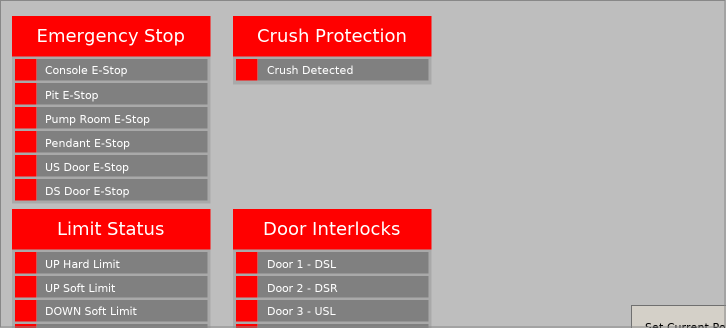
VISUALIZATION SAFETY_PANEL  // 726x328
    Rectangle (233,39 198x45)
    Rectangle (12,38 198x165)
    Rectangle (233,228 198x120)
    Rectangle (12,228 198x144)
    RoundedRectangle (15,276 21x21), colour toggle: HMI.bSoftUpLimFlag
    Rectangle (37,276 170x21)
    Rectangle (42,275 130x27), "UP Soft Limit"
    RoundedRectangle (15,300 21x21), colour toggle: HMI.bSoftDownLimFlag
    Rectangle (37,300 170x21)
    Rectangle (42,298 130x27), "DOWN Soft Limit"
    RoundedRectangle (15,324 21x21), colour variable: HMI_Hard_Limits.DownHardLimit
    Rectangle (37,324 170x21)
    Rectangle (42,322 130x27), "DOWN Hard Limit"
    RoundedRectangle (12,209 198x40), "Limit Status", colour toggle: HMI.bLimitHeaderFlag
    RoundedRectangle (236,252 21x21), colour variable: HMI_Door_Toggle.dwDoor1
    Rectangle (258,252 170x21)
    Rectangle (264,251 130x27), "Door 1 - DSL"
    RoundedRectangle (236,276 21x21), colour variable: HMI_Door_Toggle.dwDoor2
    Rectangle (258,276 170x21)
    Rectangle (264,275 130x27), "Door 2 - DSR"
    RoundedRectangle (236,300 21x21), colour variable: HMI_Door_Toggle.dwDoor3
    Rectangle (258,300 170x21)
    Rectangle (264,298 130x27), "Door 3 - USL"
    RoundedRectangle (236,324 21x21), colour variable: HMI_Door_Toggle.dwDoor4
    Rectangle (258,324 170x21)
    Rectangle (264,322 130x27), "Door 4 - USR"
    RoundedRectangle (233,209 198x40), "Door Interlocks", colour variable: HMI_Door_Toggle.dwDoorFlag
    RoundedRectangle (15,59 21x21), colour toggle: GV_LIFT.CONSOLE_ESTOP_INDICATOR_IN
    Rectangle (37,59 170x21)
    Rectangle (42,57 130x27), "Console E-Stop"
    RoundedRectangle (15,83 21x21), colour toggle: GV_LIFT.PIT_ESTOP_INDICATOR_IN
    Rectangle (37,83 170x21)
    Rectangle (42,82 130x27), "Pit E-Stop"
    RoundedRectangle (15,131 21x21), colour toggle: GV_LIFT.REMOTE_ESTOP_INDICATOR_IN
    Rectangle (37,131 170x21)
    Rectangle (42,130 130x27), "Pendant E-Stop"
    RoundedRectangle (15,155 21x21), colour toggle: GV_LIFT.UPSTAGE_ESTOP_INDICATOR_IN
    Rectangle (37,155 170x21)
    Rectangle (42,154 130x27), "US Door E-Stop"
    RoundedRectangle (12,16 198x40), "Emergency Stop", colour toggle: GV_LIFT.ESTOP_INDICATOR_OUT
    RoundedRectangle (15,179 21x21), colour toggle: GV_LIFT.DOWNSTAGE_ESTOP_INDICATOR_IN
    Rectangle (37,179 170x21)
    Rectangle (42,178 130x27), "DS Door E-Stop"
    RoundedRectangle (236,59 21x21), colour variable: HMI_Crush_Indicator.dwCrushFlag
    Rectangle (258,59 170x21)
    Rectangle (264,57 130x27), "Crush Detected"
    RoundedRectangle (233,16 198x40), "Crush Protection", colour variable: HMI_Crush_Indicator.dwCrushFlag
    Button (631,305 138x45), "Set Current Position", colour toggle: (GV_HMI.colortoggle[1])<>0
        tap GV_HMI.colortoggle[1]
        OnDialogClosed: execute { MOVE_TO_POSITION.bRecalculatePosition := TRUE; }
        OnMouseDown: write GV_HMI.updatedPos via VisuDialogs.Numpad, title 'Current Position'
    Button (631,355 138x45), "Set UP Soft Limit", colour toggle: (GV_HMI.colortoggle[2])<>0
        tap GV_HMI.colortoggle[2]
        OnMouseDown: write XML.savedvalues.UpSoftLim via VisuDialogs.Numpad, title 'Up Soft Limit'
    Button (631,405 138x45), "Set DOWN Soft Limit", colour toggle: (GV_HMI.colortoggle[3])<>0
        tap GV_HMI.colortoggle[3]
        OnMouseDown: write XML.savedvalues.DownSoftLim via VisuDialogs.Numpad, title 'Down Soft Limit'
    RoundedRectangle (15,348 21x21), colour variable: HMI_Ultimate_Limit.DownUltLimit
    Rectangle (37,348 170x21)
    Rectangle (42,346 130x27), "DOWN Ultimate Limit"
    RoundedRectangle (15,252 21x21), colour variable: HMI_Hard_Limits.UpHardLimit
    Rectangle (37,252 170x21)
    Rectangle (42,251 130x27), "UP Hard Limit"
    Rectangle (472,362 140x30), "UP Soft Limit %.2f"", text variable: XML.savedvalues.UpSoftLim
    Rectangle (472,412 140x30), "DOWN Soft Limit: %.2f"", text variable: XML.savedvalues.DownSoftLim
    RoundedRectangle (15,107 21x21), colour toggle: GV_LIFT.PUMP_ESTOP_INDICATOR_IN
    Rectangle (37,107 170x21)
    Rectangle (42,106 130x27), "Pump Room E-Stop"
END_VISUALIZATION

(* stored: Version 1.1.0.1, ProductVersion 3.1.4022.12
   Visu SAFETY_PANEL: Id {d1fbc4af-f7df-4113-9978-283b73c84b11} *)
